(* IEC 61131-3 sources: ArfBotOS/Codesys-4/ArfBotOS.fbsdev/Application.iecapp^/FUN/template/FB_Module.fb.st^/public, 5 files *)

(* ---- M_Abort.meth.st ---- *)
METHOD PUBLIC M_Abort
VAR_INPUT
END_VAR

_UnitMode.Abort();
_SeqStart := 0;  _Start:=FALSE;
_SeqHome := 0; _Home:=FALSE;
END_METHOD

(* ---- M_Hold.meth.st ---- *)
METHOD PUBLIC M_Hold
VAR_INPUT
END_VAR

_UnitMode.Hold();
END_METHOD

(* ---- M_Home.meth.st ---- *)
METHOD PUBLIC M_Home
VAR_INPUT
END_VAR

_Home:=TRUE;
END_METHOD

(* ---- M_Start.meth.st ---- *)
METHOD PUBLIC M_Start
VAR_INPUT
END_VAR

_Start := TRUE;
END_METHOD

(* ---- M_Stop.meth.st ---- *)
METHOD PUBLIC M_Stop
VAR_INPUT
END_VAR

_UnitMode.Stop();
END_METHOD
